// SIMATIC STEP 7 (V5.x) project F_ANALYS
// program: S7 Program(1)

SYMBOL_TABLE
"FAULT_ANALYS_1"	FB 145	FB 145	// Анализ отказов(T8)
END_SYMBOL_TABLE

FUNCTION_BLOCK "FAULT_ANALYS_1"	// FB 145
TITLE = Анализ гипотетических отказов двигателя
//Для анализа используем сигналы с датчиков расхода.
AUTHOR : ETSystem
VERSION : 0.1
VAR_INPUT
  FE1_PV : REAL ;
  FE2_PV : REAL ;
  FE_LIM : REAL  := 3.000000e+002;
  DELAY_T : S5TIME  := S5T#10S;
  PUMP_ON : BOOL ;
  AUTO_ON : BOOL ;
END_VAR
VAR_OUTPUT
  PAZ : BOOL ;
END_VAR
VAR
  LT_SUMM : REAL ;
END_VAR
BEGIN
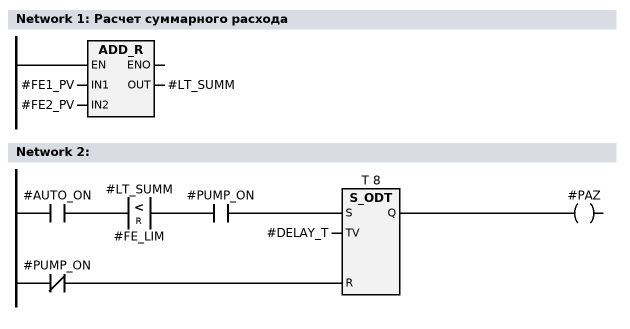
NETWORK
TITLE = Расчет суммарного расхода
      L     #FE1_PV;
      L     #FE2_PV;
      +R;
      T     #LT_SUMM;
      NOP   0;
NETWORK
TITLE =
      A     #AUTO_ON;
      A(;
      L     #LT_SUMM;
      L     #FE_LIM;
      <R;
      );
      A     #PUMP_ON;
      L     #DELAY_T;
      SD    T 8;
      AN    #PUMP_ON;
      R     T 8;
      NOP   0;
      NOP   0;
      A     T 8;
      =     #PAZ;
END_FUNCTION_BLOCK

ORGANIZATION_BLOCK OB 1
TITLE = "Main Program Sweep (Cycle)"
VERSION : 0.1
VAR_TEMP
  OB1_EV_CLASS : BYTE ;	//Bits 0-3 = 1 (Coming event), Bits 4-7 = 1 (Event class 1)
  OB1_SCAN_1 : BYTE ;	//1 (Cold restart scan 1 of OB 1), 3 (Scan 2-n of OB 1)
  OB1_PRIORITY : BYTE ;	//Priority of OB Execution
  OB1_OB_NUMBR : BYTE ;	//1 (Organization block 1, OB1)
  OB1_RESERVED_1 : BYTE ;	//Reserved for system
  OB1_RESERVED_2 : BYTE ;	//Reserved for system
  OB1_PREV_CYCLE : INT ;	//Cycle time of previous OB1 scan (milliseconds)
  OB1_MIN_CYCLE : INT ;	//Minimum cycle time of OB1 (milliseconds)
  OB1_MAX_CYCLE : INT ;	//Maximum cycle time of OB1 (milliseconds)
  OB1_DATE_TIME : DATE_AND_TIME ;	//Date and time OB1 started
END_VAR
BEGIN
// (block stored without names or comments; labels and parameter names are numbered)
END_ORGANIZATION_BLOCK
